{attribute addProperty BoxType "EL6201-0000-0017"}
{attribute addProperty Id "Slave_22A_DI0BIT10.125169Slave_22A_DI1BIT10.125170Slave_22A_DI2BIT10.125171Slave_22A_DI3BIT10.125172Slave_22B_DI0BIT10.125173Slave_22B_DI1BIT10.125174Slave_22B_DI2BIT10.125175Slave_22B_DI3BIT10.125176"}
{attribute addProperty CRC "3328292365"}
{attribute addProperty SizeInBites "8"}
{attribute addProperty SizeInBytes "1"}
TYPE Slave_22_Inputs_C661B60D :
STRUCT
	{attribute addProperty Name "Slave_22A_DI0"}
	Slave_22A_DI0 : BIT;
	{attribute addProperty Name "Slave_22A_DI1"}
	Slave_22A_DI1 : BIT;
	{attribute addProperty Name "Slave_22A_DI2"}
	Slave_22A_DI2 : BIT;
	{attribute addProperty Name "Slave_22A_DI3"}
	Slave_22A_DI3 : BIT;
	{attribute addProperty Name "Slave_22B_DI0"}
	Slave_22B_DI0 : BIT;
	{attribute addProperty Name "Slave_22B_DI1"}
	Slave_22B_DI1 : BIT;
	{attribute addProperty Name "Slave_22B_DI2"}
	Slave_22B_DI2 : BIT;
	{attribute addProperty Name "Slave_22B_DI3"}
	Slave_22B_DI3 : BIT;
END_STRUCT
END_TYPE

(* stored: Version 1.2.0.0, ProductVersion 3.1.4024.9
   DUT Slave_22_Inputs_C661B60D: Id {8c5f5af9-ad55-4eb8-8046-11e058bc732e} *)
